// TIA Portal V19 export
FUNCTION "TetraPakV70_10" : Void   // FC122, STL
TITLE = Tetra Pak V70 IO-Link DeviceID 10 Process Data
{ S7_Optimized_Access := 'TRUE' }
FAMILY : IO_Link
// Data words uses in function
// 
// HMI_CMD, dw X - command word from SCADA
// Bit 0 = auto
// Bit 1 = Manuel deactivate
// Bit 2 = Manuel activate
// Bit 3 = Locate
// Bit 4 = SV_2 Selection Bit
// Bit 5 = SV_3 Selection Bit
// Bit 6 = spare
// 
// HMI_INFO, dw X - info word to SCADA
// Bit 0  = activated
// Bit 1  = changing
// Bit 2  = faulty 
// Bit 3  = auto_man, Manual = 1 
// Bit 4  = man_on_off
// Bit 5  = Reset_FB
// Bit 6  = ManualSelected
// Bit 7  = Set_FB
// Bit 8  = Locate Active 
// Bit 9  = TrippedInd
// Bit 10 = IsolatedInd
// Bit 11 = VSD_Fault 
// Bit 12 = VSD_Alarm
// Bit 13 = sv_3Activated
// Bit 14 = fb_error - Alarm feedback error
// Bit 15 = sv_2Activated  
// 
// Error status
// 0 (Everything is OK)
// 16 (Sensor target missing (#16))
// 17 (Setup prerequisite issue (#17))
// 18 (Pneumatic part issue (#18))
// 19 (Seat lift sensor issue (#19))
// 20 (Position not reached (#20))
// 21 (Unexpected movement (#21))
// 22 (Seat-lift sensor missing (#22))
// 23 (Pilot valve 1 missing (#23))
// 24 (Pilot valve 2 missing (#24))
// 25 (Pilot valve 3 missing (#25))
// 26 (Interlock active (#26))
// 27 (Output short circuit (#27))
// 28 (Setup aborted (#28))
// 29 (Blocked button (#29))
// 30 (Communication failure (#30))
// 31 (Safety stop active (#31))
// stored: AutoNumber false
   VAR_INPUT
      Addr : Int;   // First Byte address of 4 byte address space
      Pulse : Bool;   // Trigger one clean pulse on SV_1
      Burst : Bool;   // Enable burst clean
      SV_1 : Bool;   // Trigger solenoid valve 1 for main valve activation
      SV_2 : Bool;   // Trigger solenoid valve 2 for upper seat lift activation
      SV_3 : Bool;   // Trigger solenoid valve 3 for lower seat push activation
      Wink : Bool;   // Visual indictation for locating the unit
   END_VAR
   VAR_OUTPUT
      ValvePosition : Real;   // Current Valve Position (0 - 1060 * 0.1)
      ValveState : Bool;   // Current Valve State
      O_DI4 : Bool;   // Output signal status Pin 4
      O_DI2 : Bool;   // Output signal status Pin 2
      Teach : Bool;   // Teach output for teach command bit
   END_VAR
   VAR_IN_OUT
      itemInfo : "ItemInfo_UDT";
      itemCommand : "ItemCommand_UDT";
      ErrorStatus : Byte;   // See Block Comment
      LSP : Bool;   // Lower Seat Push energised position
      USL : Bool;   // Upper Seat Lift energised position
      Main : Bool;   // Main energised position
      DE_EN : Bool;   // De-energised
      O_DA : Bool;   // Output device recognised
      O_DE : Bool;   // Output device error event has appeared
      O_PQ : Bool;   // Output port qualifer proces data valid
   END_VAR
   VAR_TEMP
      TW_Flag : Word;
      Tmp_ErrorStatus : Byte;   // Local Byte 6
      output : Bool;
      sv1_out : Bool;
      sv2_out : Bool;
      sv3_out : Bool;
   END_VAR
BEGIN

NETWORK
TITLE = info to scada, free
// L     #HMI_INFO
// Get first byte address
      L     #Addr;
      SLW   3;
      LAR1;
// **************  Inputs *******************
// Valve Position
      L     IW [AR1, P#0.0];
      DTR;
      L     0.1;
      *R;
      T     #ValvePosition;

// Error Status
      L     IB [AR1, P#2.0];
      T     #Tmp_ErrorStatus;
      SET;
      R     #Tmp_ErrorStatus.%X5;
      R     #Tmp_ErrorStatus.%X6;
      R     #Tmp_ErrorStatus.%X7;
      L     #Tmp_ErrorStatus;
      T     #ErrorStatus;


// ValveState
      L     IB [AR1, P#3.0];
      T     #TW_Flag;
      L     16;
      AW;
      L     16;
      ==I;
      =     #ValveState;

// LSP
      L     IB [AR1, P#3.0];
      T     #TW_Flag;
      L     4;
      AW;
      L     4;
      ==I;
      =     #LSP;

// USL
      L     IB [AR1, P#3.0];
      T     #TW_Flag;
      L     3;
      AW;
      L     3;
      ==I;
      =     #USL;

// Main
      L     IB [AR1, P#3.0];
      T     #TW_Flag;
      L     2;
      AW;
      L     2;
      ==I;
      =     #Main;

// DE_EN
      L     IB [AR1, P#3.0];
      T     #TW_Flag;
      L     1;
      AW;
      L     1;
      ==I;
      =     #DE_EN;

// PQI

      L     IB [AR1, P#4.0];
      T     #TW_Flag;

      L     #TW_Flag;
      L     1;
      AW;
      L     1;
      ==I;
      =     #O_DI4;



      L     #TW_Flag;
      L     2;
      AW;
      L     2;
      ==I;
      =     #O_DI2;

      L     #TW_Flag;
      L     32;
      AW;
      L     32;
      ==I;
      =     #O_DA;

      L     #TW_Flag;
      L     64;
      AW;
      L     64;
      ==I;
      =     #O_DE;


      L     #TW_Flag;
      L     128;
      AW;
      L     128;
      ==I;
      =     #O_PQ;

// *** Valve Fault Detected ***
      L     #ErrorStatus;
      L     1;
      >I;
      O;
      A     #O_DE;
      O;
      AN    #O_DA;
      AN    #O_DE;
      AN    #O_PQ;
      =     #itemInfo.fb_error;

// Pulse
      A     #Pulse;
      =     Q [AR1, P#0.2];  // Pulse output

// Burst
      A     #Burst;
      =     Q [AR1, P#0.3];

// Valve Control
      SET;
      R     #sv1_out;
      R     #sv2_out;
      R     #sv3_out;

      A     #SV_1;
      AN    #itemInfo.auto_man;  // IF AUTO
      O(;
      A     #itemInfo.auto_man;  // IF Manual
      AN    #itemCommand.SV_2SelectionBit;
      AN    #itemCommand.SV_3SelectionBit;
      A     #itemInfo.man_on_off;  // Manual on/off
      );
      JCN   sv2;
      =     #sv1_out;

sv2:  A     #SV_2;
      AN    #itemInfo.auto_man;  // IF AUTO
      O(;
      A     #itemInfo.auto_man;  // IF Manual
      A     #itemCommand.SV_2SelectionBit;
      AN    #itemCommand.SV_3SelectionBit;
      A     #itemInfo.man_on_off;  // Manual on/off
      );
      JCN   sv3;
      =     #sv2_out;

sv3:  A     #SV_3;
      AN    #itemInfo.auto_man;  // IF AUTO
      O(;
      A     #itemInfo.auto_man;  // IF Manual
      AN    #itemCommand.SV_2SelectionBit;
      A     #itemCommand.SV_3SelectionBit;
      A     #itemInfo.man_on_off;  // Manuel on/off
      );
      JCN   svx;
      =     #sv3_out;

svx:  A     #sv1_out;
      O     #sv2_out;
      O     #sv3_out;
      =     #output;

      A     #sv1_out;
      =     Q [AR1, P#0.4];  // Set/reset Output
      A     #sv2_out;
      =     Q [AR1, P#0.5];  // Set/reset Output
      A     #sv3_out;
      =     Q [AR1, P#0.6];  // Set/reset Output

// Locate

      A     #itemCommand.Locate;
      A     #itemInfo.LocateActive;
      R     Q [AR1, P#0.7];
      R     #itemCommand.Locate;


      A     #itemCommand.Locate;
      AN    #itemInfo.LocateActive;
      S     Q [AR1, P#0.7];
      R     #itemCommand.Locate;

// Teach
      A     #itemCommand.Teach;
      =     #Teach;

//****************** Outputs ************

      L     QB [AR1, P#0.0];
      T     QB [AR1, P#0.0];




NETWORK
TITLE = SCADA INFO & command
      AN    #itemCommand.Locate;
      AN    #itemCommand.Man_Act;
      AN    #itemCommand.Man_DeAct;
      AN    #itemCommand.Teach;
      AN    #itemCommand.SpareBool;
      AN    #itemCommand.SpareBool_1;
      AN    #itemCommand.SpareBool_2;
      AN    #itemCommand.SpareBool_3;
      AN    #itemCommand.SpareBool_4;
      AN    #itemCommand.SpareBool_5;
      AN    #itemCommand.SpareBool_6;
      AN    #itemCommand.SpareBool_7;
      AN    #itemCommand.SV_2SelectionBit;
      AN    #itemCommand.SV_3SelectionBit;
      AN    #itemCommand.SpareBool_10;
      JC    INFO;  // if commamd bits = 0 then no commands


      A     #itemCommand.Auto;
      R     #itemInfo.auto_man;
      JC    clea;

      A     #itemCommand.Man_DeAct;
      S     #itemInfo.auto_man;
      R     #itemInfo.man_on_off;
      JC    clea;

      A     #itemCommand.Man_Act;
      S     #itemInfo.auto_man;
      S     #itemInfo.man_on_off;
      JC    clea;
// Clear itemCommand word
clea: SET;
      R     #itemCommand.Auto;
      R     #itemCommand.Locate;
      R     #itemCommand.Man_Act;
      R     #itemCommand.Man_DeAct;
      R     #itemCommand.Teach;
      R     #itemCommand.SpareBool;
      R     #itemCommand.SpareBool_1;
      R     #itemCommand.SpareBool_2;
      R     #itemCommand.SpareBool_3;
      R     #itemCommand.SpareBool_4;
      R     #itemCommand.SpareBool_5;
      R     #itemCommand.SpareBool_6;
      R     #itemCommand.SpareBool_7;
      R     #itemCommand.SpareBool_10;

//;=========================== Scada info ================================
INFO: A     #itemInfo.fb_error;  // feedback error
      =     #itemInfo.faulty;
      A     #itemInfo.auto_man;
      =     #itemInfo.ManualSelected;  //Show Manual selected on SCADA
      A     #DE_EN;
      =     #itemInfo.Reset_FB;  //Show Reset FB in "Item Info & Operation" popup
      A     #Main;
      =     #itemInfo.Set_FB;  //Show Set FB in "Item Info & Operation" popup
      A     #LSP;
      =     #itemInfo.sv_2Activated;
      A     #USL;
      =     #itemInfo.sv_3Activated;
      A     Q [AR1, P#0.7];
      =     #itemInfo.LocateActive;


//;                     // ================================
//;                     // = SET FB , SET/RES FB = ****SV_2 FB and SV_3 FB added****
// Goto Changing
      A     #output;  // IF Output
      A     #Main;  // AND SetFB
      JC    ACT;  // Goto Activated

      A     #output;  // IF Output
      AN    #DE_EN;  // AND NOT SetFB
      JC    CHAN;

      JU    DEAC;



//;                     // ================================
//;                     // ================================
DEAC: R     #itemInfo.activated;  // Update = deactivated
      R     #itemInfo.sv_2Activated;
      R     #itemInfo.sv_3Activated;
      R     #itemInfo.changing;
      JU    NEX4;  //NEXT;
//;                     // ================================
CHAN: R     #itemInfo.activated;  // Update = activated
      R     #itemInfo.sv_2Activated;  // Update = sv2activated
      R     #itemInfo.sv_3Activated;  // Update = sv3activated
      S     #itemInfo.changing;
      JU    NEX4;  //NEXT;
//;                     // ================================
ACT:  S     #itemInfo.activated;  // Update = activated
      R     #itemInfo.changing;
      JU    NEX4;  //NEXT;


NEX4: NOP   0;
      A     #output;  // IF Output
      A     #LSP;  // AND LowerSeatFB
      JC    LACT;  // Goto LowerSeatActivated
      A     #output;  // IF Output
      A     #USL;  // AND UpperSeatFB
      JC    UACT;  // Goto UpperSeatActivated
      JU    NEX5;


//;                     // ================================
LACT: S     #itemInfo.sv_2Activated;

      JU    NEX5;
//;                     // ================================
UACT: S     #itemInfo.sv_3Activated;

      JU    NEX5;
NEX5: NOP   0;



END_FUNCTION
